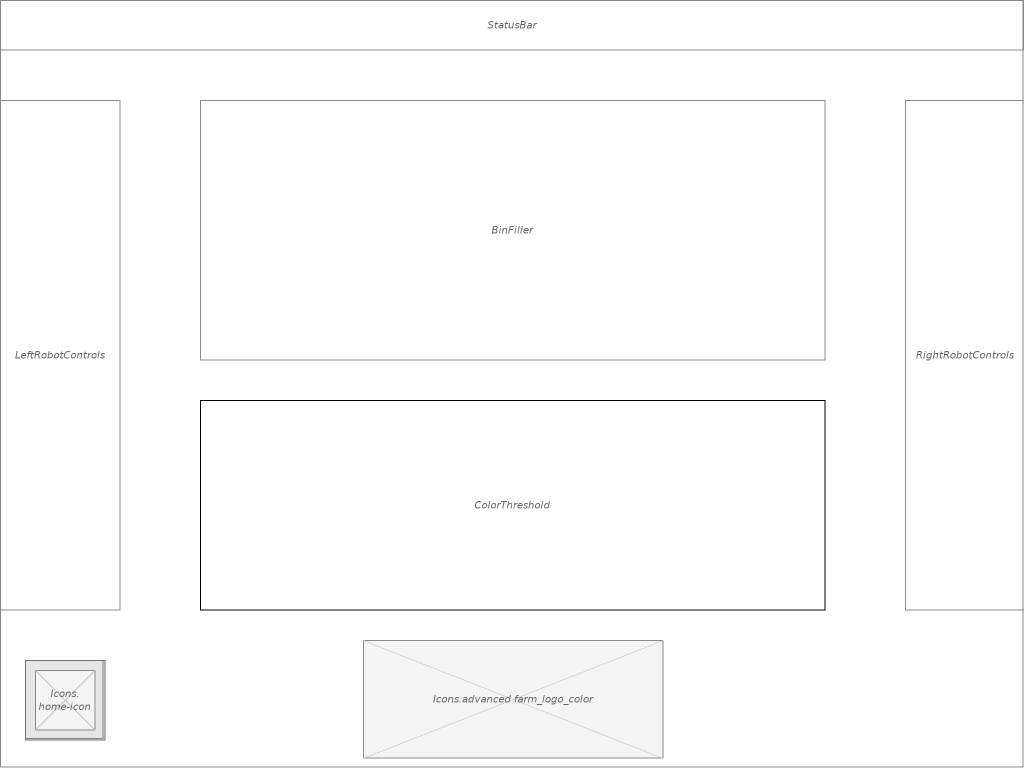
VISUALIZATION Supervisor_Screen  // 1024x768
    Frame (0,0 1024x50)
        shows StatusBar()
    Group (25,660 80x80)
        OnMouseClick: change screen: Home_Screen
        Button (0,0 80x80)
        Image (10,10 60x60), image: Icons.home-icon
    Image (363,640 300x118), image: Icons.advanced farm_logo_color
    Rectangle (200,100 625x260)
    Rectangle (905,100 120x510)
    Rectangle (0,100 120x510)
    Frame (0,100 120x510)
        shows LeftRobotControls()
    Frame (905,100 120x510)
        shows RightRobotControls()
    Frame (200,400 625x210)
        shows ColorThreshold()
    Frame (200,100 625x260)
        shows BinFiller()
    Rectangle (200,400 625x210)
END_VISUALIZATION

(* stored: Version 1.1.0.1, ProductVersion 3.1.4024.15
   Visu Supervisor_Screen: Id {41f6fd09-bc5e-4ef0-a95c-d5451c2d7621} *)
